FUNCTION DINT_TO_SIZE : ST_SIZE
VAR_INPUT
	nValue : DINT;
END_VAR

DINT_TO_SIZE.nValue := DINT_TO_UDINT(MAX(0, nValue));

END_FUNCTION

(* stored: Version 1.1.0.1, ProductVersion 3.1.4024.15
   POU DINT_TO_SIZE: Id {ddc3b84f-bb2f-4c78-ba03-d96cfdee9268}, SpecialFunc None *)
